Fanuc KAREL source: compact_preamble.KL

PROGRAM KB00123
%NOLOCKGROUP
%ENVIRONMENT FDEV
VAR
P1 : STRING[80];P2:INTEGER
BEGIN
P1='A'
P2=1
MOVE_FILE(P1,P2)
END KB00123
